// 1-WORD divide to 2-USINT
FUNCTION WORD_TO_USINT_Bit : outWord
VAR_INPUT
	nOutput : WORD;
END_VAR
VAR
	outWord : outWord;
END_VAR

outWord.Lower := TO_USINT(nOutput); //Lower Bits
outWord.Upper := TO_USINT(SHR(nOutput, 8)); //Uppper Bits
WORD_TO_USINT_Bit := outWord;

END_FUNCTION

(* stored: Version 1.1.0.1, ProductVersion 3.1.4024.12
   POU WORD_TO_USINT_Bit: Id {d74012c4-c5d6-4668-9e8c-027d00f76e1b}, SpecialFunc None *)
